# EPICS substitutions: apps/plcApp/Db/solenoid_mps_addons.substitutions
file "db/torus_ai_renamed.db" {
    pattern { P R PV PLCID TAG EGU PREC }
{ B_SOL: MPS: TP8630 PLC_SOL TP8630 K 2 }
{ B_SOL: MPS: TP8631 PLC_SOL TP8631 K 2 }
{ B_SOL: MPS: TP8632 PLC_SOL TP8632 K 2 }
}
